// Mitsubishi GX Works2 project: TIMERS   PLC: Q02/Q02H

PROGRAM MAIN
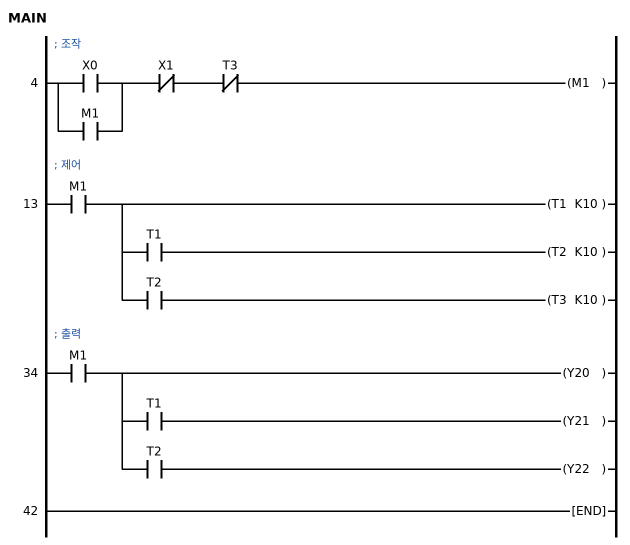
; 조작
4     LD      X0
      OR      M1
      ANI     X1
      ANI     T3
      OUT     M1
; 제어
13    LD      M1
      OUT     T1 K10
      MPS
      AND     T1
      OUT     T2 K10
      MPP
      AND     T2
      OUT     T3 K10
; 출력
34    LD      M1
      OUT     Y20
      MPS
      AND     T1
      OUT     Y21
      MPP
      AND     T2
      OUT     Y22
42    END
END_PROGRAM

PROGRAM FLASH
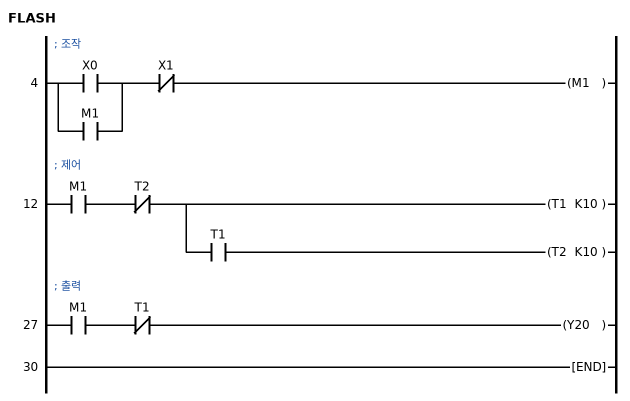
; 조작
4     LD      X0
      OR      M1
      ANI     X1
      OUT     M1
; 제어
12    LD      M1
      ANI     T2
      OUT     T1 K10
      AND     T1
      OUT     T2 K10
; 출력
27    LD      M1
      ANI     T1
      OUT     Y20
30    END
END_PROGRAM

PROGRAM TIMER
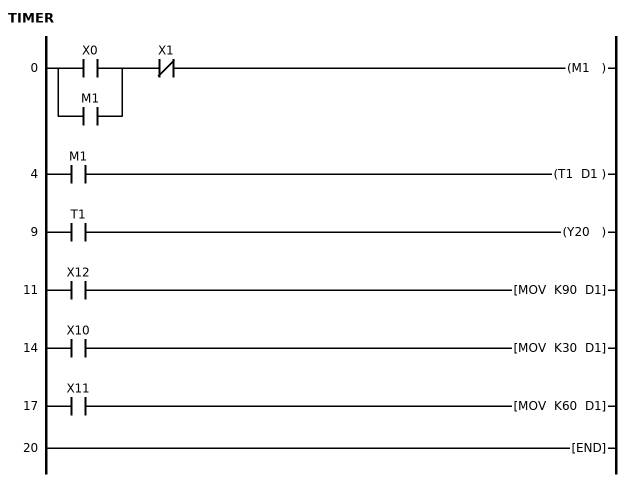
0     LD      X0
      OR      M1
      ANI     X1
      OUT     M1
4     LD      M1
      OUT     T1 D1
9     LD      T1
      OUT     Y20
11    LD      X12
      MOV     K90 D1
14    LD      X10
      MOV     K30 D1
17    LD      X11
      MOV     K60 D1
20    END
END_PROGRAM

PROGRAM CLK
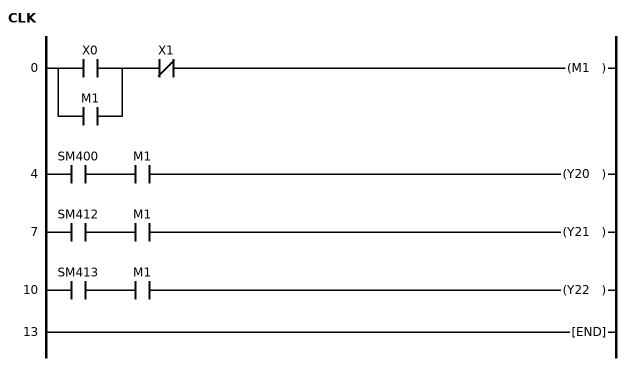
0     LD      X0
      OR      M1
      ANI     X1
      OUT     M1
4     LD      SM400
      AND     M1
      OUT     Y20
7     LD      SM412
      AND     M1
      OUT     Y21
10    LD      SM413
      AND     M1
      OUT     Y22
13    END
END_PROGRAM

PROGRAM STAIR4
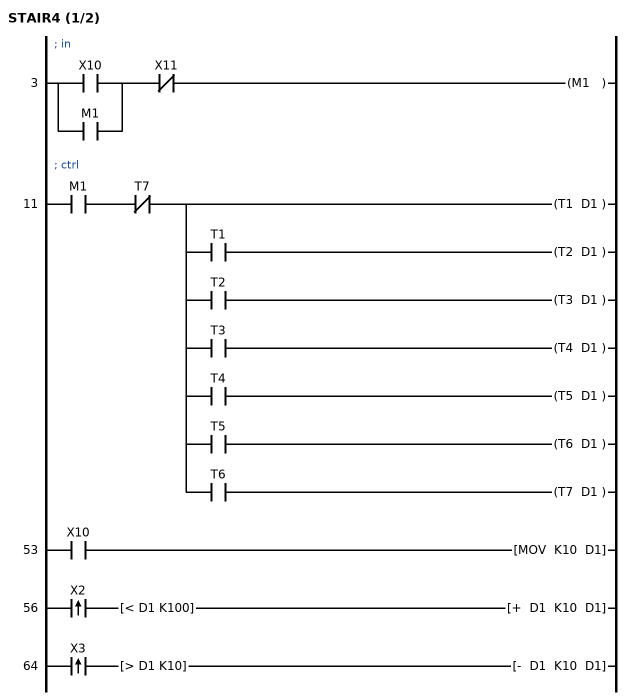
; in
3     LD      X10
      OR      M1
      ANI     X11
      OUT     M1
; ctrl
11    LD      M1
      ANI     T7
      OUT     T1 D1
      MPS
      AND     T1
      OUT     T2 D1
      MRD
      AND     T2
      OUT     T3 D1
      MRD
      AND     T3
      OUT     T4 D1
      MRD
      AND     T4
      OUT     T5 D1
      MRD
      AND     T5
      OUT     T6 D1
      MPP
      AND     T6
      OUT     T7 D1
53    LD      X10
      MOV     K10 D1
56    LDP     X2
      AND<    D1 K100
      +       D1 K10 D1
64    LDP     X3
      AND>    D1 K10
      -       D1 K10 D1
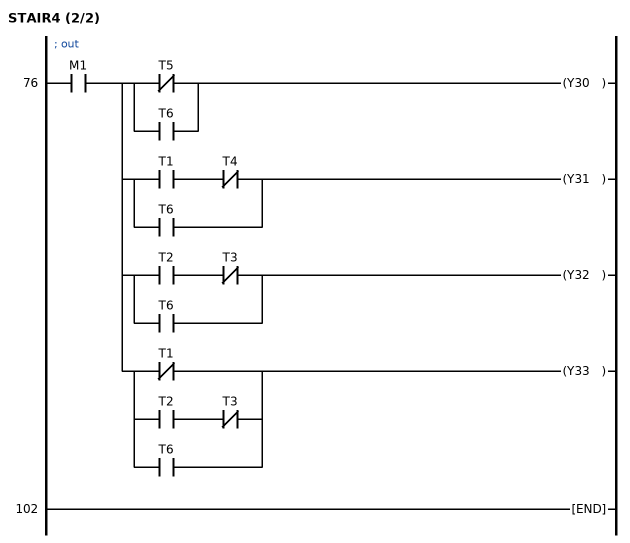
; out
76    LD      M1
      MPS
      LDI     T5
      OR      T6
      ANB
      OUT     Y30
      MRD
      LD      T1
      ANI     T4
      OR      T6
      ANB
      OUT     Y31
      MRD
      LD      T2
      ANI     T3
      OR      T6
      ANB
      OUT     Y32
      MPP
      LDI     T1
      LD      T2
      ANI     T3
      ORB
      OR      T6
      ANB
      OUT     Y33
102   END
END_PROGRAM

PROGRAM STAIR2
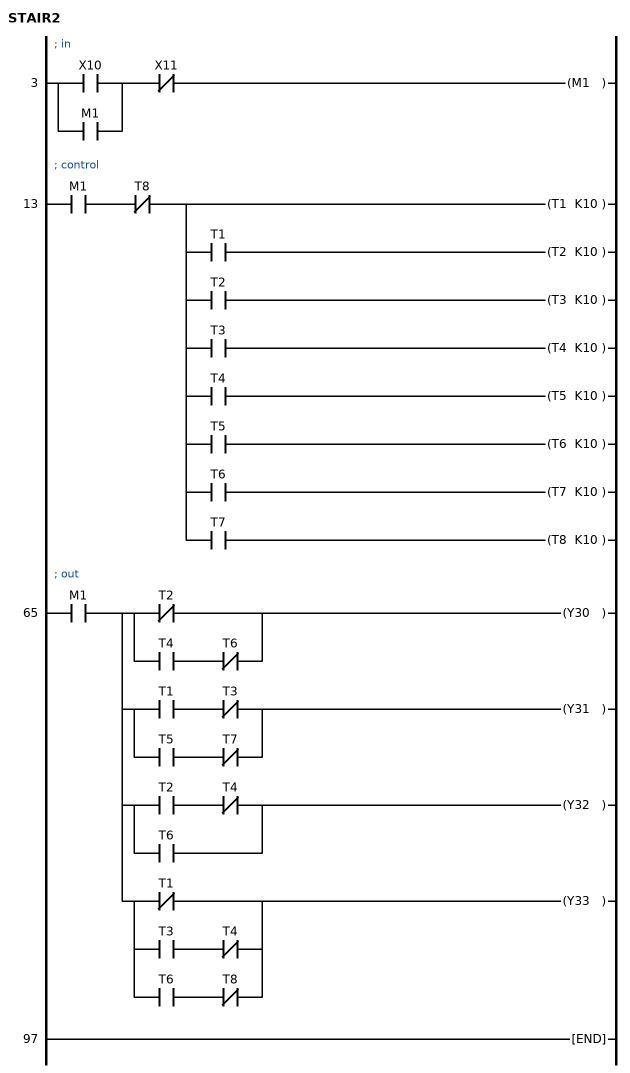
; in
3     LD      X10
      OR      M1
      ANI     X11
      OUT     M1
; control
13    LD      M1
      ANI     T8
      OUT     T1 K10
      MPS
      AND     T1
      OUT     T2 K10
      MRD
      AND     T2
      OUT     T3 K10
      MRD
      AND     T3
      OUT     T4 K10
      MRD
      AND     T4
      OUT     T5 K10
      MRD
      AND     T5
      OUT     T6 K10
      MRD
      AND     T6
      OUT     T7 K10
      MPP
      AND     T7
      OUT     T8 K10
; out
65    LD      M1
      MPS
      LDI     T2
      LD      T4
      ANI     T6
      ORB
      ANB
      OUT     Y30
      MRD
      LD      T1
      ANI     T3
      LD      T5
      ANI     T7
      ORB
      ANB
      OUT     Y31
      MRD
      LD      T2
      ANI     T4
      OR      T6
      ANB
      OUT     Y32
      MPP
      LDI     T1
      LD      T3
      ANI     T4
      ORB
      LD      T6
      ANI     T8
      ORB
      ANB
      OUT     Y33
97    END
END_PROGRAM

PROGRAM PULSETIM
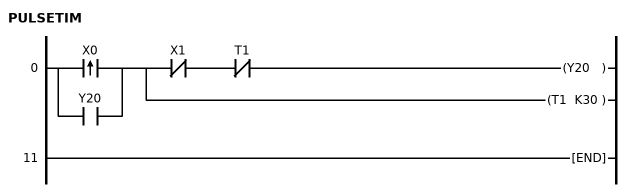
0     LDP     X0
      OR      Y20
      MPS
      ANI     X1
      ANI     T1
      OUT     Y20
      MPP
      OUT     T1 K30
11    END
END_PROGRAM

PROGRAM STAIR3
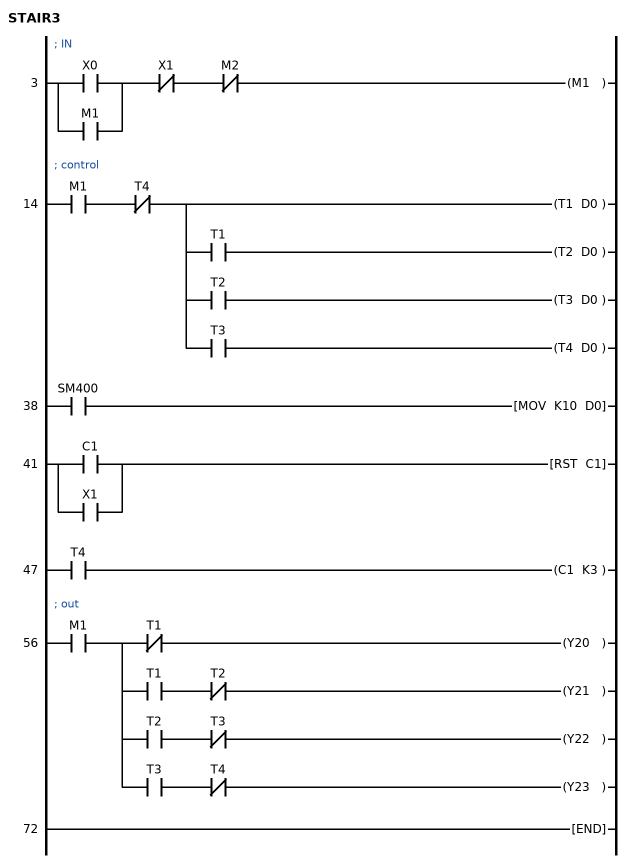
; IN
3     LD      X0
      OR      M1
      ANI     X1
      ANI     M2
      OUT     M1
; control
14    LD      M1
      ANI     T4
      OUT     T1 D0
      MPS
      AND     T1
      OUT     T2 D0
      MRD
      AND     T2
      OUT     T3 D0
      MPP
      AND     T3
      OUT     T4 D0
38    LD      SM400
      MOV     K10 D0
41    LD      C1
      OR      X1
      RST     C1
47    LD      T4
      OUT     C1 K3
; out
56    LD      M1
      MPS
      ANI     T1
      OUT     Y20
      MRD
      AND     T1
      ANI     T2
      OUT     Y21
      MRD
      AND     T2
      ANI     T3
      OUT     Y22
      MPP
      AND     T3
      ANI     T4
      OUT     Y23
72    END
END_PROGRAM
